(*
  Systron camera system
  Provides callback function (rx_callback) for received TcpIp messages.   
*)
FUNCTION_BLOCK FB_SystronCamera EXTENDS FB_CameraTcpIp

VAR
  stCameraResult            : ARRAY [1..cNbCameras] OF ST_CAMERA_RESULT;

  nNbTrigger                : INT;
END_VAR

VAR CONSTANT                
  cNbCameras                : UDINT := 2;                (*Number of Systron cameras*)

  cErrorString              : T_MaxString := '<Error(';
  cStartString              : T_MaxString := '<position(';
  cEndingString             : T_MaxString := ');';

  cCameraMinXY              : REAL := -20.0;  (*[mm]*)
  cCameraMaxXY              : REAL := +20.0;  (*[mm]*)
END_VAR

(*Simulation*)
IF _bSimulate THEN
  CreateSimCamPoints();
END_IF

(*
  Simulate camera data
*)
METHOD CreateSimCamPoints : BOOL
VAR_INST
  fbTonTimer    : TON;    (*Send timer*)
  nCounter      : UDINT;  (*Loop counter*)
END_VAR
(*Test points*)
stCameraResult[1].x_ref :=   54;  (*[mm]*)
stCameraResult[1].y_ref := 1003;  (*[mm]*)
stCameraResult[1].valid := TRUE;
stCameraResult[2].x_ref :=   46;  (*[mm]*)
stCameraResult[2].y_ref :=  376;  (*[mm]*)
stCameraResult[2].valid := TRUE;

(*Points are send every 15s*)
fbTonTimer(IN := NOT fbTonTimer.Q, PT := T#15S);
IF fbTonTimer.Q THEN
  FOR nCounter := 1 TO 2 DO
    stCamPoint.x_ref := F_MeterToSubPixelReal( stCameraResult[nCounter].x_ref * 0.001      (*[mm] => [m]*)
                                             , UDINT_TO_LREAL(_nPrintUnitResolution));     (*Result should be in pixels*)
    stCamPoint.y_ref := F_MeterToSubPixelReal( stCameraResult[nCounter].y_ref * 0.001      (*[m]*)
                                             , UDINT_TO_LREAL(_nPrintUnitResolution));     (*Result should be in pixels*)
    stCamPoint.dx    := F_MeterToSubPixelReal( 0.100 * UDINT_TO_REAL(nCounter) * 0.001     (*[mm] => [m]*)
                                            , UDINT_TO_LREAL(_nPrintUnitResolution));     (*Result should be in pixels*)
    stCamPoint.dy    := F_MeterToSubPixelReal( 0.200 * UDINT_TO_REAL(nCounter) * 0.001     (*[mm] => [m]*)
                                            , UDINT_TO_LREAL(_nPrintUnitResolution));     (*Result should be in pixels*)
  
    _iCameraSink.AddCamPoint(stCamPoint);
  END_FOR  
END_IF
END_METHOD

{attribute 'monitoring':='call'}
PROPERTY eCameraMode : E_CameraMode
GET
eCameraMode := _eCameraMode;
IF _eCameraMode = E_CameraMode.Auto THEN
  eCameraMode := E_CameraMode.XYR;
END_IF
END_GET
END_PROPERTY

PROPERTY eDeviceType : E_CameraDevice
GET
eDeviceType := E_CameraDevice.PrintMark;
END_GET
END_PROPERTY

METHOD GetCamStatus : BOOL
VAR_OUTPUT
  bConnectionOK  : BOOL;    // Camera connected
  bTeachOk       : BOOL;    // Teach successful
  nTeachedPoints : UDINT;   // Teached points for this job
  nScannedPoints : UDINT;   // Scanned points on current sheet
  bCamStarted    : BOOL;    // Camera trigger is active, cam started
  bCamDone       : BOOL;    // Camera finished on last CT
  bErrors        : ARRAY[1..GVL_Camera.nC_NbCamErrors] OF BOOL;  // generic error flag list
END_VAR
bConnectionOK  := NOT bConnectionErr OR bSimulate;
bTeachOk       := TRUE; //NO teach availabe (teached by a specific sheet from machine)
nTeachedPoints := 0;
nScannedPoints := 0;
bCamStarted    := _bCamTriggerStarted;
bCamDone       := _bCamTriggerDone; 
{warning 'TODO: get real teach information'}

GetCamStatus := bConnectionOK;
END_METHOD

METHOD rx_callback
VAR_INPUT
	sMessage	: CalmarCompTcpIp.ST_TcpMsg;
END_VAR

VAR
  sAnalyzeLastMessage    : T_MaxString;          (*telegram string*)

  nCounter               : UDINT;
  nFindIndex             : INT;
END_VAR
SUPER^.rx_callback(sMessage := sMessage);

sAnalyzeLastMessage := sLastMessage;

nFindIndex := FIND(sAnalyzeLastMessage, cErrorString);
IF nFindIndex > 0 THEN
  (*Error received*)
  sLastErrorMessage := (DELETE(sAnalyzeLastMessage, (nFindIndex + LEN(cErrorString) - 1), 1));

  (*Extract error message*)
  nFindIndex := FIND(sLastErrorMessage, cEndingString);
  IF nFindIndex > 0 THEN
    sLastErrorMessage := (DELETE(sLastErrorMessage, LEN(sLastErrorMessage) - nFindIndex, nFindIndex));
  END_IF;
ELSE
  (*Search for start string*)
  nFindIndex := FIND(sAnalyzeLastMessage, cStartString);
  IF nFindIndex > 0 THEN
    (*Search string found => remove string to generate index*)
    sAnalyzeLastMessage := (DELETE(sAnalyzeLastMessage, (nFindIndex + LEN(cStartString) - 1), 1));

    (*Search for trigger number*)
    nFindIndex := FIND(sAnalyzeLastMessage, ',');
    IF nFindIndex > 0 THEN
      nNbTrigger := STRING_TO_INT(LEFT(sAnalyzeLastMessage, (nFindIndex - 1)));

      sAnalyzeLastMessage := (DELETE(sAnalyzeLastMessage, nFindIndex, 1));
    END_IF;

    (*Search for rx, ry, v, x and y*)
    FOR nCounter := 1 TO cNbCameras DO
      stCameraResult[nCounter].valid := TRUE;

      (*rx*)
      nFindIndex := FIND(sAnalyzeLastMessage, ',');
      IF nFindIndex > 0 THEN
        stCameraResult[nCounter].x_ref := STRING_TO_REAL(LEFT(sAnalyzeLastMessage, (nFindIndex - 1)));

        IF    (stCameraResult[nCounter].x_ref < cCameraMinXY)
           OR (stCameraResult[nCounter].x_ref > cCameraMaxXY)
        THEN
          stCameraResult[nCounter].valid := FALSE;
        END_IF;

        sAnalyzeLastMessage := (DELETE(sAnalyzeLastMessage, nFindIndex, 1));
      ELSE
        stCameraResult[nCounter].valid := FALSE;
      END_IF;
      (*ry*)
      nFindIndex := FIND(sAnalyzeLastMessage, ',');
      IF nFindIndex > 0 THEN
        stCameraResult[nCounter].y_ref := STRING_TO_REAL(LEFT(sAnalyzeLastMessage, (nFindIndex - 1)));

        IF    (stCameraResult[nCounter].y_ref < cCameraMinXY)
           OR (stCameraResult[nCounter].y_ref > cCameraMaxXY)
        THEN
          stCameraResult[nCounter].valid := FALSE;
        END_IF;

        sAnalyzeLastMessage := (DELETE(sAnalyzeLastMessage, nFindIndex, 1));
      ELSE
        stCameraResult[nCounter].valid := FALSE;
      END_IF;
      (*v*)
      nFindIndex := FIND(sAnalyzeLastMessage, ',');
      IF nFindIndex > 0 THEN
        IF FIND(LEFT(sAnalyzeLastMessage, (nFindIndex - 1)), 'True') > 0 THEN
          stCameraResult[nCounter].valid := TRUE;
        ELSE
          stCameraResult[nCounter].valid := FALSE;
        END_IF;

        sAnalyzeLastMessage := (DELETE(sAnalyzeLastMessage, nFindIndex, 1));
      ELSE
        stCameraResult[nCounter].valid := FALSE;
      END_IF;
      (*x*)
      nFindIndex := FIND(sAnalyzeLastMessage, ',');
      IF nFindIndex > 0 THEN
        stCameraResult[nCounter].x := STRING_TO_REAL(LEFT(sAnalyzeLastMessage, (nFindIndex - 1)));

        IF    (stCameraResult[nCounter].x < cCameraMinXY)
           OR (stCameraResult[nCounter].x > cCameraMaxXY)
        THEN
          stCameraResult[nCounter].valid := FALSE;
        END_IF;

        sAnalyzeLastMessage := (DELETE(sAnalyzeLastMessage, nFindIndex, 1));
      ELSE
        stCameraResult[nCounter].valid := FALSE;
      END_IF;
      (*y*)
      nFindIndex := FIND(sAnalyzeLastMessage, ',');
      IF nFindIndex > 0 THEN
        stCameraResult[nCounter].y := STRING_TO_REAL(LEFT(sAnalyzeLastMessage, (nFindIndex - 1)));

        IF    (stCameraResult[nCounter].y < cCameraMinXY)
           OR (stCameraResult[nCounter].y > cCameraMaxXY)
        THEN
          stCameraResult[nCounter].valid := FALSE;
        END_IF;

        sAnalyzeLastMessage := (DELETE(sAnalyzeLastMessage, nFindIndex, 1));
      ELSE
        nFindIndex := FIND(sAnalyzeLastMessage, ')');
        IF nFindIndex > 0 THEN
          stCameraResult[nCounter].y := STRING_TO_REAL(LEFT(sAnalyzeLastMessage, (nFindIndex - 1)));

          IF    (stCameraResult[nCounter].y < cCameraMinXY)
             OR (stCameraResult[nCounter].y > cCameraMaxXY)
          THEN
            stCameraResult[nCounter].valid := FALSE;
          END_IF;

          sAnalyzeLastMessage := (DELETE(sAnalyzeLastMessage, nFindIndex, 1));
        ELSE
          stCameraResult[nCounter].valid := FALSE;
        END_IF;
      END_IF;
    END_FOR;
  ELSE
    (*Search string not found*)
    FOR nCounter := 1 TO cNbCameras DO
      stCameraResult[nCounter].valid := FALSE;
    END_FOR;
  END_IF;
END_IF;

IF _iCameraSink <> 0 THEN
  FOR nCounter := 1 TO cNbCameras DO
    stCamPoint.x_ref := F_MeterToSubPixelReal( stCameraResult[nCounter].x_ref * 0.001              (*[mm] => [m]*)
                                         , UDINT_TO_LREAL(_nPrintUnitResolution));             (*Result should be in pixels*)
    stCamPoint.y_ref := F_MeterToSubPixelReal( stCameraResult[nCounter].y_ref * 0.001              (*[m]*)
                                         , UDINT_TO_LREAL(_nPrintUnitResolution));             (*Result should be in pixels*)
    stCamPoint.dx    := F_MeterToSubPixelReal( (stCameraResult[nCounter].x_ref - stCameraResult[nCounter].x) * 0.001  (*[mm] => [m]*)
                                         , UDINT_TO_LREAL(_nPrintUnitResolution));             (*Result should be in pixels*)
    stCamPoint.dy    := F_MeterToSubPixelReal( (stCameraResult[nCounter].y_ref - stCameraResult[nCounter].y) * 0.001  (*[mm] => [m]*)
                                         , UDINT_TO_LREAL(_nPrintUnitResolution));             (*Result should be in pixels*)

    _iCameraSink.AddCamPoint(stCamPoint);
  END_FOR
END_IF;

bMsgReceived := FALSE;
END_METHOD

(*
  Set mode to camera.
  :return: TRUE if success
*)
METHOD setCameraMode : BOOL
VAR_INPUT
  eCameraMode : E_CameraMode;
END_VAR
IF eCameraMode = E_CameraMode.NoCorrection OR  // supported modi
   eCameraMode = E_CameraMode.XYR THEN
 
  _eCameraMode := eCameraMode;  // set desired mode
  setCameraMode := TRUE;
ELSE
  LogError(F_Concat3('Camera mode=', TO_STRING(eCameraMode), ' not supported by camera'));
  _eCameraMode := E_CameraMode.NoCorrection;
END_IF
END_METHOD

{attribute 'monitoring':='variable'}
PROPERTY sName : STRING
GET
sName := 'Systron';
END_GET
END_PROPERTY

END_FUNCTION_BLOCK

(* stored: Version 1.1.0.1, ProductVersion 3.1.4024.9
   POU FB_SystronCamera: Id {a6c36bce-dec5-430c-b3a6-e5194ad905ad}, SpecialFunc None
   Method CreateSimCamPoints: Id {378225cb-fa44-4cef-9044-ea9afe88fa30}
   Property eCameraMode: Id {e5951198-b845-45c0-92a9-897b5e1419fe}
   Get Get: Id {b2d1200e-b7cd-4992-9f8e-c57d8aa4d63b}
   Property eDeviceType: Id {fd11a3fc-8283-45e9-999a-5c5324ba9a9d}
   Get Get: Id {762cc984-2f98-4132-8053-db984330df56}
   Method GetCamStatus: Id {9304763a-bd41-4825-aaf3-90140932f9d8}
   Method rx_callback: Id {2340d0b0-adae-46c1-9b1b-c4b18a35dcd3}
   Method setCameraMode: Id {720266e4-d8ef-40ae-b05d-dc2210fe930e}
   Property sName: Id {b04a7b8e-bad3-4516-bd51-f585d8c1b504}
   Get Get: Id {875f39da-3007-4bc5-9d85-8922d38e9eac} *)
